// TIA Portal V20 export
DATA_BLOCK "Config"   // DB14
{ DB_Accessible_From_OPC_UA := 'FALSE' }
AUTHOR : ERsystem_FA2_DH. Kim
// stored: Access Published, DBAccessibleFromOPCUA false, DBAccessibleFromWebserver false, MemoryReserve 100, Namespace Unit1.Em0
   VAR RETAIN
      em { ExternalWritable := 'False'} : "LAF_typeEmConfiguration";
      axis { ExternalAccessible := 'False'; ExternalVisible := 'False'; ExternalWritable := 'False'} : Array[1.._.U1EM0_NO_OF_AXES] of DB_ANY;
      cmUnwinderTopAxisB { ExternalAccessible := 'False'; ExternalVisible := 'False'; ExternalWritable := 'False'} : "LBC_typeAxis64PosConfiguration";
      cmAirShaftTopOnOff { ExternalAccessible := 'False'; ExternalVisible := 'False'; ExternalWritable := 'False'} : "LBC_typeTwoWayActuatorConfiguration";
      cmRadiusMeasureTop { ExternalAccessible := 'False'; ExternalVisible := 'False'; ExternalWritable := 'False'} : "LBC_typeAnalogInputConfiguration";
      cmEpcTop { ExternalAccessible := 'False'; ExternalVisible := 'False'; ExternalWritable := 'False'} : "LER_typeCON600Configuration";
      cmTopDirectionCheckSensor { S7_SetPoint := 'True'} : "LBC_typeDigitalSignalConfiguration";
      cmRadiusMeasure : "LER_typeRadiusMeasureConfiguration";
      softCam : Struct
         unwinderTopAxisB : "LER_typeSoftCamInterface";
      END_STRUCT;
      Data : Array[0..10] of LReal;
   END_VAR
BEGIN
   em.referenceDesignator.parent := WSTRING#'U1';
   em.referenceDesignator.relative := WSTRING#'EM0 SepaUnwinderTop';
   em.referenceDesignator.combined := WSTRING#'U1.EM0 SepaUnwinderTop';
   axis[1] := 85;
   axis[2] := 364;
   cmUnwinderTopAxisB.referenceDesignator := WSTRING#'UnwinderTopAxisB';
   cmAirShaftTopOnOff.referenceDesignator := WSTRING#'cmAirShaftTopOnOff';
   cmAirShaftTopOnOff.monitoringLeavingFeedback := T#500MS;
   cmAirShaftTopOnOff.monitoringReachingFeedback := T#500MS;
   cmAirShaftTopOnOff.monitoringDiscrepancy := T#0MS;
   cmAirShaftTopOnOff.setOutputHomeContinuously := TRUE;
   cmAirShaftTopOnOff.setOutputWorkContinuously := TRUE;
   cmAirShaftTopOnOff.disableHomeCommand := FALSE;
   cmAirShaftTopOnOff.disableFeedbackHomePos := TRUE;
   cmAirShaftTopOnOff.disableFeedbackWorkPos := TRUE;
   cmAirShaftTopOnOff.disableAlarms := FALSE;
   cmAirShaftTopOnOff.resetOutputsOnError := FALSE;
   cmAirShaftTopOnOff.allwaysWaitOnReachingTime := FALSE;
   cmRadiusMeasureTop.referenceDesignator := WSTRING#'cmTopRadiusMeasure';
   cmRadiusMeasureTop.physicalUnit := 'mm';
   cmRadiusMeasureTop.isUnipolarSignal := TRUE;
   cmRadiusMeasureTop.default := 0.0;
   cmRadiusMeasureTop.limitHigh2 := 400.0;
   cmRadiusMeasureTop.limitHigh1 := 200.0;
   cmRadiusMeasureTop.limitLow1 := -200.0;
   cmRadiusMeasureTop.limitLow2 := -400.0;
   cmRadiusMeasureTop.processValueMax := 400.0;
   cmRadiusMeasureTop.processValueMin := 0.0;
   cmRadiusMeasureTop.scaleAnalogUppPoint := 27670.0;
   cmRadiusMeasureTop.scaleAnalogLowPoint := 0.0;
   cmRadiusMeasureTop.scaleProcessUppPoint := 180.0;
   cmRadiusMeasureTop.scaleProcessLowPoint := 0.0;
   cmRadiusMeasureTop.disableAlarms := TRUE;
   cmTopDirectionCheckSensor.referenceDesignator := WSTRING#'cmTopDirectionCheckSensor';
   cmTopDirectionCheckSensor.onDelay := T#0MS;
   cmTopDirectionCheckSensor.offDelay := T#0MS;
   cmTopDirectionCheckSensor.default := FALSE;
   cmTopDirectionCheckSensor.invertProcessValue := FALSE;
   cmTopDirectionCheckSensor.disableAlarms := FALSE;
   cmRadiusMeasure.Offset := 39.0;
   cmRadiusMeasure.DecimalPoint := 1;
END_DATA_BLOCK
